TYPE MDP5001_342_066CA8C6 :
STRUCT
	MDP5001_342_Input	: MDP5001_342_I_066CA8C6;
	MDP5001_342_Output	: MDP5001_342_O_066CA8C6;
END_STRUCT
END_TYPE

(* stored: Version 1.1.0.1, ProductVersion 3.1.4024.12
   DUT MDP5001_342_066CA8C6: Id {b528fd1a-8abb-4abb-ad76-d81cea84189e} *)
